Staubli VAL3: txtBoxDynUpdate.pgx

public program txtBoxDynUpdate(string x_sDynamicText)
begin
  // This program updates the dynamic text of a text box message
  //
  // Input param
  // x_nDynamicText    : Dynamic part of the message
  //
  //
  // Created 23-02-05                           C.CURRIVAND
  //------------------------------------------------------------------
  call strAlign(x_sDynamicText,nTxtBoxWidth,"L"," ")
  call type(nTxtBoxCol+1,nTxtBoxRow+size(sWrkString),x_sDynamicText)
end
